(* Schneider Machine Expert - Basic project pick_place_SCADA, file version 2.7.0.0 *)
(* ProjectInformations: Name=New project *)

HARDWARE
  Cpu 0: TM221C16R
  EthernetConfiguration: NetworkName=M221, IpAllocationMode=FixedAddress, IpAddress=0.0.0.0, SubnetMask=0.0.0.0
  SerialLineConfiguration: Baud=Baud19200, Parity=ParityEven, DataBits=DataBits8, StopBits=StopBits1, PhysicalMedium=PhysicalMediumRs485, TransmissionMode=TransmissionModeModbusRtu, SlaveId=1, Addressing=SlaveAddressing
  MastTask: UsePeriodScanMode=false, PeriodScan=100
  FastTask: Period=255
  CpuBehavior: StartingMode=StartAsPreviousState, AutoSaveRamOnEeprom=true, WatchdogPeriod=250

SYMBOLS  (address, symbol, comment, settings)
  %M0       BOX_AT_PLACE
  %M1       PART_AT_PLACE
  %M2       DETECTED
  %M3       C_LIMIT
  %M4       START_
  %M5       RESET
  %M6       STOP
  %M7       EMERGENCY_STOP
  %M8       AUTO
  %M10      SENSOR_SALIDA
  %M20      BOX_CONVEYOR
  %M21      PART_CONVEYOR
  %M22      EXIT_CONVEYOR
  %M23      C_MAS
  %M24      GRAB
  %M25      EXIT_GREEN
  %M26      EXIT_YELLOW
  %M27      EXIT_RED
  %M28      START_LIGHT
  %M29      RESET_LIGHT
  %M30      STOP_LIGHT
  %M31      BOX_EMITTER
  %M32      PART_EMITTER
  %M33      FACTORY_RESET
  %M34      REMOVE
  %M50      GRAB_SCADA
  %M52      GIRO_ARDUINO
  %M54      STOP_ARDUINO
  %M56      RESET_ARDUINO
  %M60      E0
  %M61      E1
  %M62      E2
  %M63      E3
  %M64      E4
  %M65      E5
  %M66      E6
  %M67      E7
  %M68      E8
  %M69      E9
  %M70      E10
  %M71      E11
  %M72      E12
  %M77      E1_1
  %M80      E_MANUAL
  %M81      E3_1
  %M82      E7_1
  %M90      C1
  %M91      C2
  %MD0      X
  %MD2      Y
  %MD4      Z
  %MD10     SP_X
  %MD12     SP_Y
  %MD14     SP_Z
  %MD16     COUNTER
  %MD18     DISPLAY_PEDIDO
  %MD26     SP_X_ARDUINO
  %MD28     SP_Y_SCADA
  %MD30     SP_Z_SCADA
  %MD32     PEDIDO_ARDUINO
  %TM0      TON_1  [Preset=2, Base=OneSecond]
  %TM1      TON_2  [Preset=2, Base=OneSecond]
  %TM2      TON_3  [Preset=2, Base=OneSecond]
  %TM3        [Preset=1, Base=OneSecond]
  %TM4        [Preset=1, Base=OneSecond]
  %TM5        [Preset=3, Base=OneSecond]
  %TM6        [Preset=2, Base=OneSecond]
  %TM7        [Preset=2, Base=OneSecond]
  %TM8        [Preset=2, Base=OneSecond]

POU New POU
  (* SectionNumber=1 *)

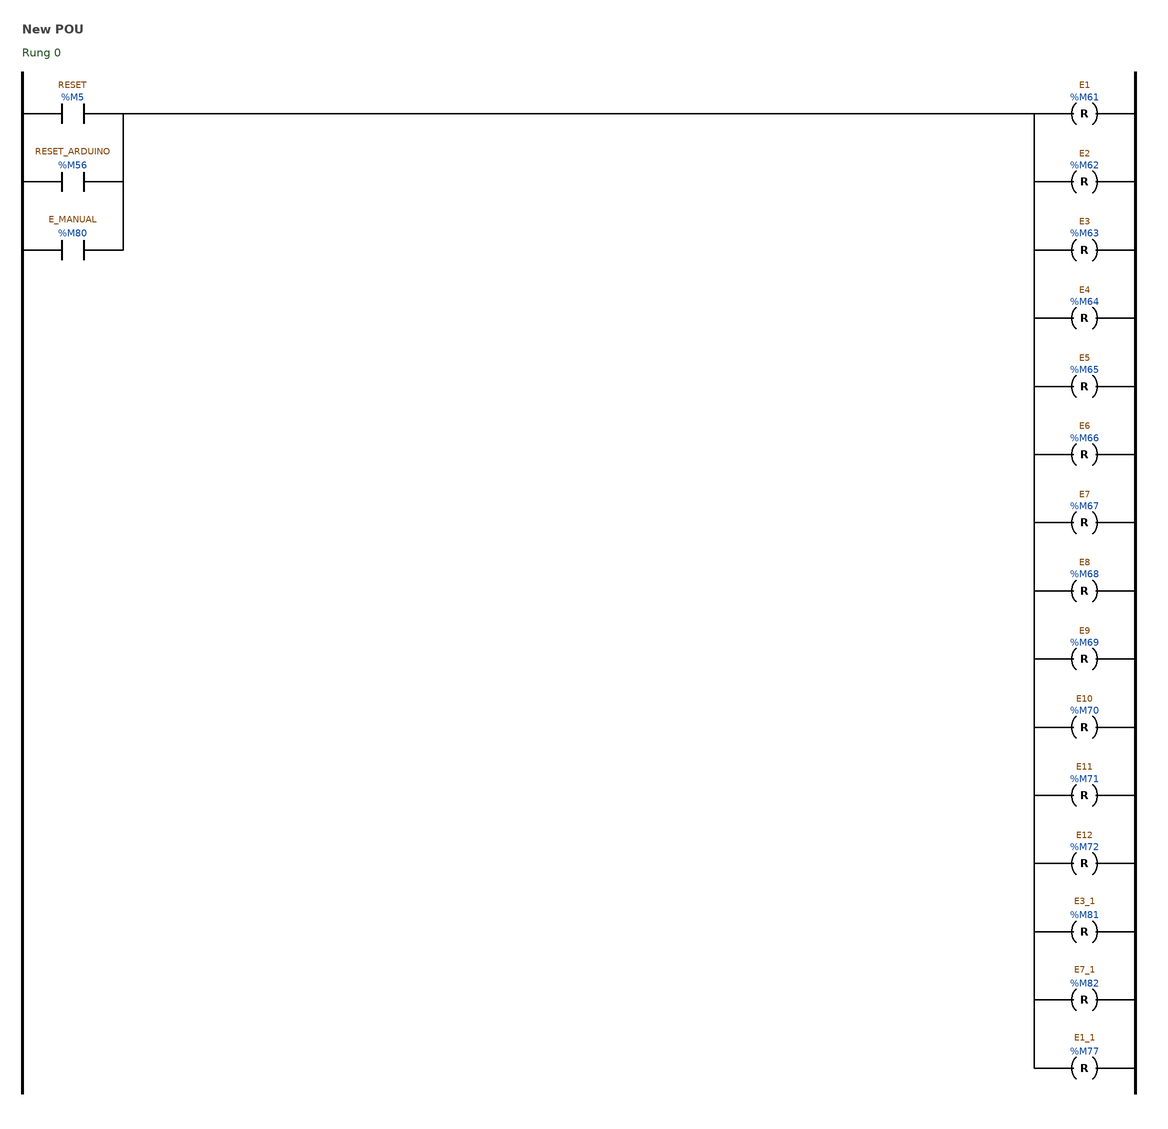

// Rung 0
  LD %M5                  (* RESET *)
  OR %M56                 (* RESET_ARDUINO *)
  OR %M80                 (* E_MANUAL *)
  R %M61                  (* E1 *)
  R %M62                  (* E2 *)
  R %M63                  (* E3 *)
  R %M64                  (* E4 *)
  R %M65                  (* E5 *)
  R %M66                  (* E6 *)
  R %M67                  (* E7 *)
  R %M68                  (* E8 *)
  R %M69                  (* E9 *)
  R %M70                  (* E10 *)
  R %M71                  (* E11 *)
  R %M72                  (* E12 *)
  R %M81                  (* E3_1 *)
  R %M82                  (* E7_1 *)
  R %M77                  (* E1_1 *)
  // as ST:
  //   IF RESET OR RESET_ARDUINO OR E_MANUAL THEN E1 := FALSE; END_IF;
  //   IF RESET OR RESET_ARDUINO OR E_MANUAL THEN E2 := FALSE; END_IF;
  //   IF RESET OR RESET_ARDUINO OR E_MANUAL THEN E3 := FALSE; END_IF;
  //   IF RESET OR RESET_ARDUINO OR E_MANUAL THEN E4 := FALSE; END_IF;
  //   IF RESET OR RESET_ARDUINO OR E_MANUAL THEN E5 := FALSE; END_IF;
  //   IF RESET OR RESET_ARDUINO OR E_MANUAL THEN E6 := FALSE; END_IF;
  //   IF RESET OR RESET_ARDUINO OR E_MANUAL THEN E7 := FALSE; END_IF;
  //   IF RESET OR RESET_ARDUINO OR E_MANUAL THEN E8 := FALSE; END_IF;
  //   IF RESET OR RESET_ARDUINO OR E_MANUAL THEN E9 := FALSE; END_IF;
  //   IF RESET OR RESET_ARDUINO OR E_MANUAL THEN E10 := FALSE; END_IF;
  //   IF RESET OR RESET_ARDUINO OR E_MANUAL THEN E11 := FALSE; END_IF;
  //   IF RESET OR RESET_ARDUINO OR E_MANUAL THEN E12 := FALSE; END_IF;
  //   IF RESET OR RESET_ARDUINO OR E_MANUAL THEN E3_1 := FALSE; END_IF;
  //   IF RESET OR RESET_ARDUINO OR E_MANUAL THEN E7_1 := FALSE; END_IF;
  //   IF RESET OR RESET_ARDUINO OR E_MANUAL THEN E1_1 := FALSE; END_IF;

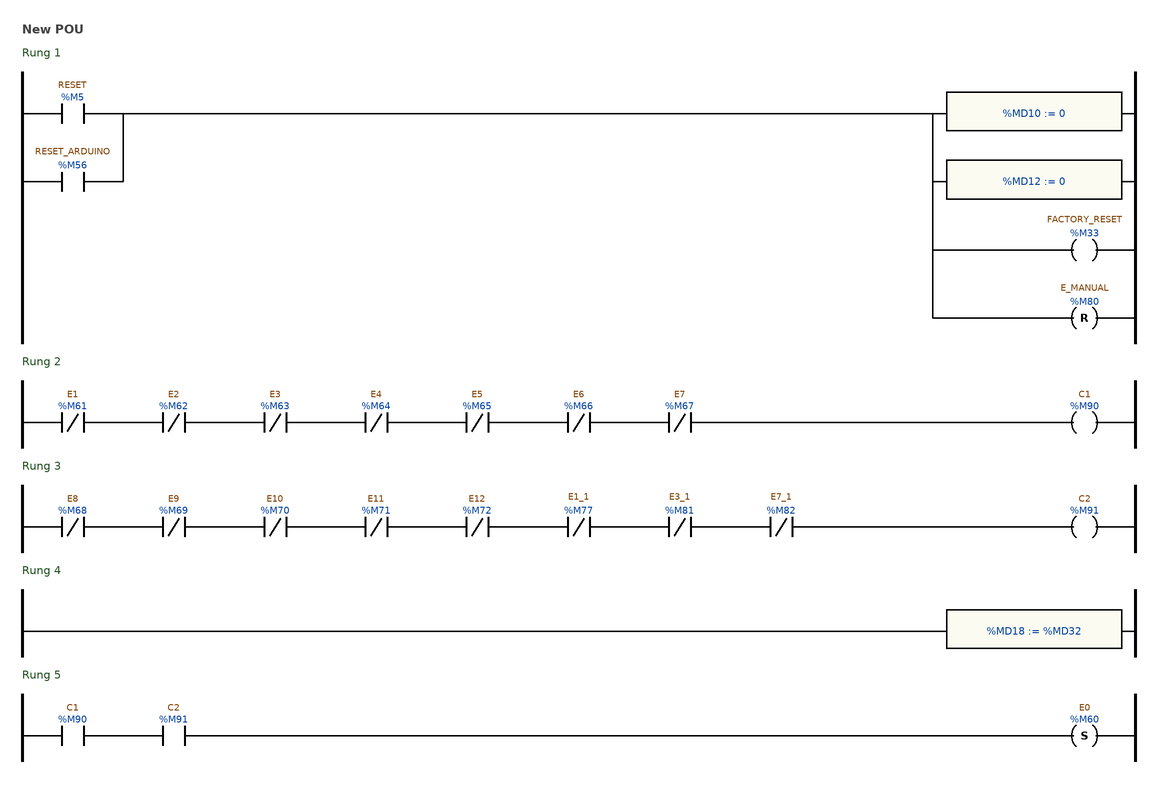

// Rung 1
  LD %M5                  (* RESET *)
  OR %M56                 (* RESET_ARDUINO *)
  [ %MD10 := 0 ]          (* SP_X *)
  [ %MD12 := 0 ]          (* SP_Y *)
  ST %M33                 (* FACTORY_RESET *)
  R %M80                  (* E_MANUAL *)
  // as ST:
  //   IF RESET OR RESET_ARDUINO THEN SP_X := 0; END_IF;
  //   IF RESET OR RESET_ARDUINO THEN SP_Y := 0; END_IF;
  //   FACTORY_RESET := RESET OR RESET_ARDUINO;
  //   IF RESET OR RESET_ARDUINO THEN E_MANUAL := FALSE; END_IF;

// Rung 2
  LDN %M61                (* E1 *)
  ANDN %M62               (* E2 *)
  ANDN %M63               (* E3 *)
  ANDN %M64               (* E4 *)
  ANDN %M65               (* E5 *)
  ANDN %M66               (* E6 *)
  ANDN %M67               (* E7 *)
  ST %M90                 (* C1 *)
  // as ST:
  //   C1 := NOT E1 AND NOT E2 AND NOT E3 AND NOT E4 AND NOT E5 AND NOT E6 AND NOT E7;

// Rung 3
  LDN %M68                (* E8 *)
  ANDN %M69               (* E9 *)
  ANDN %M70               (* E10 *)
  ANDN %M71               (* E11 *)
  ANDN %M72               (* E12 *)
  ANDN %M77               (* E1_1 *)
  ANDN %M81               (* E3_1 *)
  ANDN %M82               (* E7_1 *)
  ST %M91                 (* C2 *)
  // as ST:
  //   C2 := NOT E8 AND NOT E9 AND NOT E10 AND NOT E11 AND NOT E12 AND NOT E1_1 AND NOT E3_1 AND NOT E7_1;

// Rung 4
  LD 1
  [ %MD18 := %MD32 ]      (* DISPLAY_PEDIDO, PEDIDO_ARDUINO *)
  // as ST:
  //   DISPLAY_PEDIDO := PEDIDO_ARDUINO;

// Rung 5
  LD %M90                 (* C1 *)
  AND %M91                (* C2 *)
  S %M60                  (* E0 *)
  // as ST:
  //   IF C1 AND C2 THEN E0 := TRUE; END_IF;

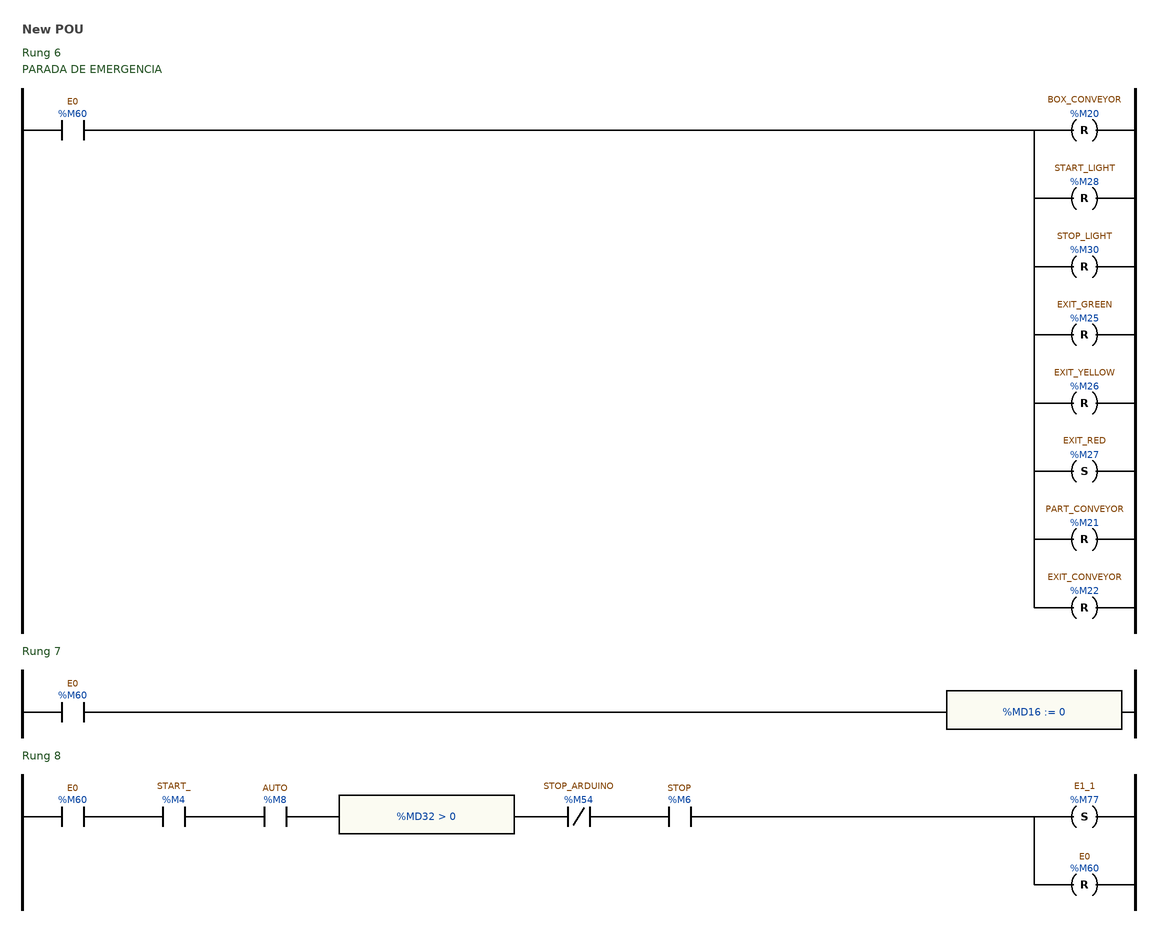

// Rung 6
// PARADA DE EMERGENCIA
  LD %M60                 (* E0 *)
  R %M20                  (* BOX_CONVEYOR *)
  R %M28                  (* START_LIGHT *)
  R %M30                  (* STOP_LIGHT *)
  R %M25                  (* EXIT_GREEN *)
  R %M26                  (* EXIT_YELLOW *)
  S %M27                  (* EXIT_RED *)
  R %M21                  (* PART_CONVEYOR *)
  R %M22                  (* EXIT_CONVEYOR *)
  // as ST:
  //   IF E0 THEN BOX_CONVEYOR := FALSE; END_IF;
  //   IF E0 THEN START_LIGHT := FALSE; END_IF;
  //   IF E0 THEN STOP_LIGHT := FALSE; END_IF;
  //   IF E0 THEN EXIT_GREEN := FALSE; END_IF;
  //   IF E0 THEN EXIT_YELLOW := FALSE; END_IF;
  //   IF E0 THEN EXIT_RED := TRUE; END_IF;
  //   IF E0 THEN PART_CONVEYOR := FALSE; END_IF;
  //   IF E0 THEN EXIT_CONVEYOR := FALSE; END_IF;

// Rung 7
  LD %M60                 (* E0 *)
  [ %MD16 := 0 ]          (* COUNTER *)
  // as ST:
  //   IF E0 THEN COUNTER := 0; END_IF;

// Rung 8
  LD %M60                 (* E0 *)
  AND %M4                 (* START_ *)
  AND %M8                 (* AUTO *)
  AND [ %MD32 > 0 ]       (* PEDIDO_ARDUINO *)
  ANDN %M54               (* STOP_ARDUINO *)
  AND %M6                 (* STOP *)
  S %M77                  (* E1_1 *)
  R %M60                  (* E0 *)
  // as ST:
  //   IF E0 AND START_ AND AUTO AND PEDIDO_ARDUINO > 0 AND NOT STOP_ARDUINO AND STOP THEN E1_1 := TRUE; END_IF;
  //   IF E0 AND START_ AND AUTO AND PEDIDO_ARDUINO > 0 AND NOT STOP_ARDUINO AND STOP THEN E0 := FALSE; END_IF;

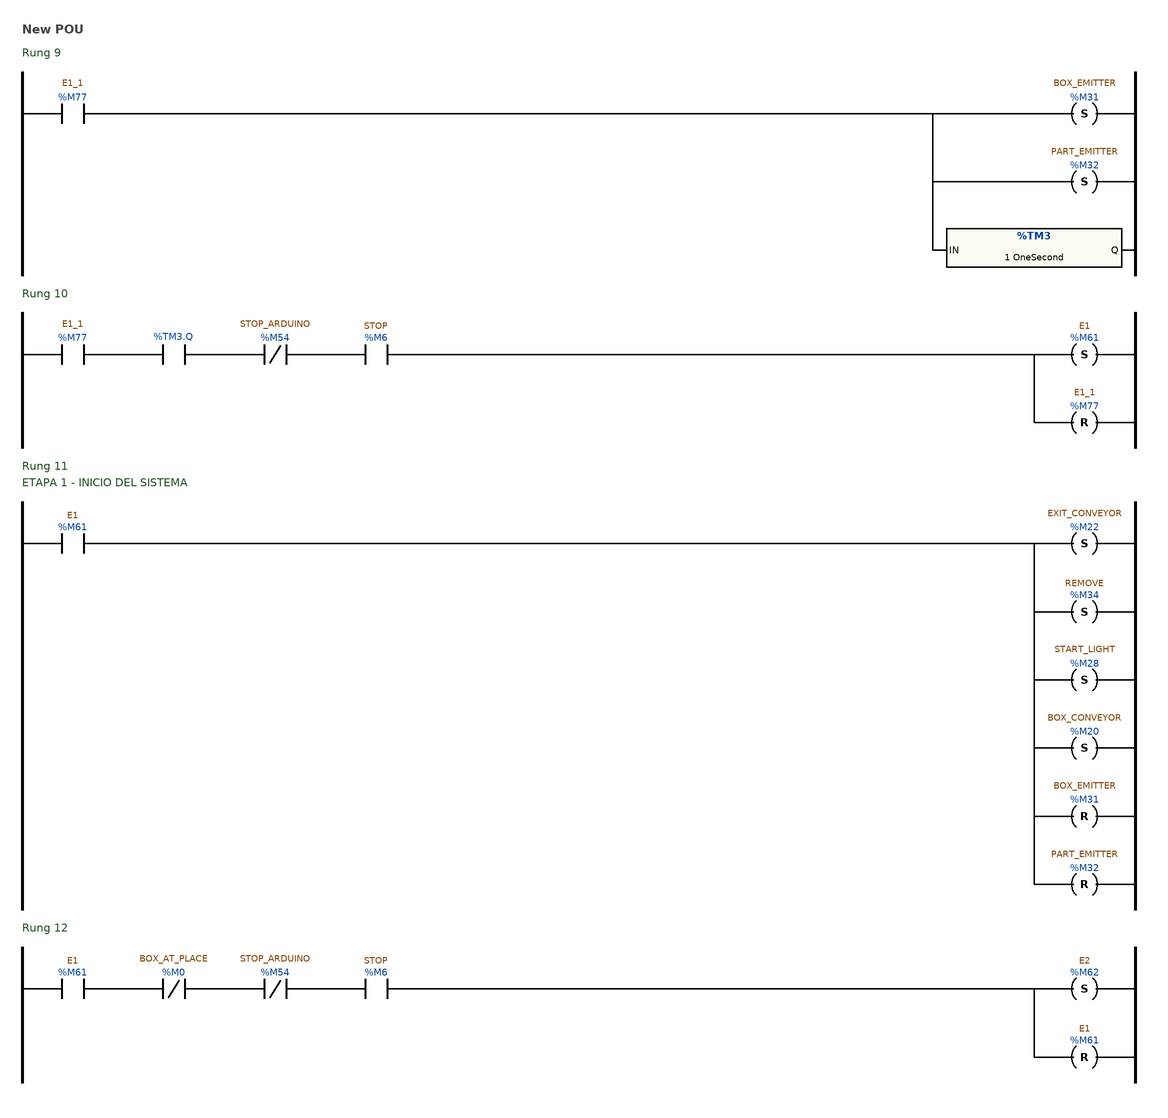

// Rung 9
  LD 1
  MULTIFB
  LD 1
  AND %M77                (* E1_1 *)
  ST %MW2009:X0
  LD %MW2009:X0
  S %M31                  (* BOX_EMITTER *)
  S %M32                  (* PART_EMITTER *)
  BLK %TM3
  LD %MW2009:X0
  IN
  END_BLK
  MULTIFB
  // as ST:
  //   IF E1_1 THEN BOX_EMITTER := TRUE; END_IF;
  //   IF E1_1 THEN PART_EMITTER := TRUE; END_IF;
  //   %TM3(IN := E1_1);

// Rung 10
  LD %M77                 (* E1_1 *)
  AND %TM3.Q
  ANDN %M54               (* STOP_ARDUINO *)
  AND %M6                 (* STOP *)
  S %M61                  (* E1 *)
  R %M77                  (* E1_1 *)
  // as ST:
  //   IF E1_1 AND %TM3.Q AND NOT STOP_ARDUINO AND STOP THEN E1 := TRUE; END_IF;
  //   IF E1_1 AND %TM3.Q AND NOT STOP_ARDUINO AND STOP THEN E1_1 := FALSE; END_IF;

// Rung 11
// ETAPA 1 - INICIO DEL SISTEMA
  LD %M61                 (* E1 *)
  S %M22                  (* EXIT_CONVEYOR *)
  S %M34                  (* REMOVE *)
  S %M28                  (* START_LIGHT *)
  S %M20                  (* BOX_CONVEYOR *)
  R %M31                  (* BOX_EMITTER *)
  R %M32                  (* PART_EMITTER *)
  // as ST:
  //   IF E1 THEN EXIT_CONVEYOR := TRUE; END_IF;
  //   IF E1 THEN REMOVE := TRUE; END_IF;
  //   IF E1 THEN START_LIGHT := TRUE; END_IF;
  //   IF E1 THEN BOX_CONVEYOR := TRUE; END_IF;
  //   IF E1 THEN BOX_EMITTER := FALSE; END_IF;
  //   IF E1 THEN PART_EMITTER := FALSE; END_IF;

// Rung 12
  LD %M61                 (* E1 *)
  ANDN %M0                (* BOX_AT_PLACE *)
  ANDN %M54               (* STOP_ARDUINO *)
  AND %M6                 (* STOP *)
  S %M62                  (* E2 *)
  R %M61                  (* E1 *)
  // as ST:
  //   IF E1 AND NOT BOX_AT_PLACE AND NOT STOP_ARDUINO AND STOP THEN E2 := TRUE; END_IF;
  //   IF E1 AND NOT BOX_AT_PLACE AND NOT STOP_ARDUINO AND STOP THEN E1 := FALSE; END_IF;

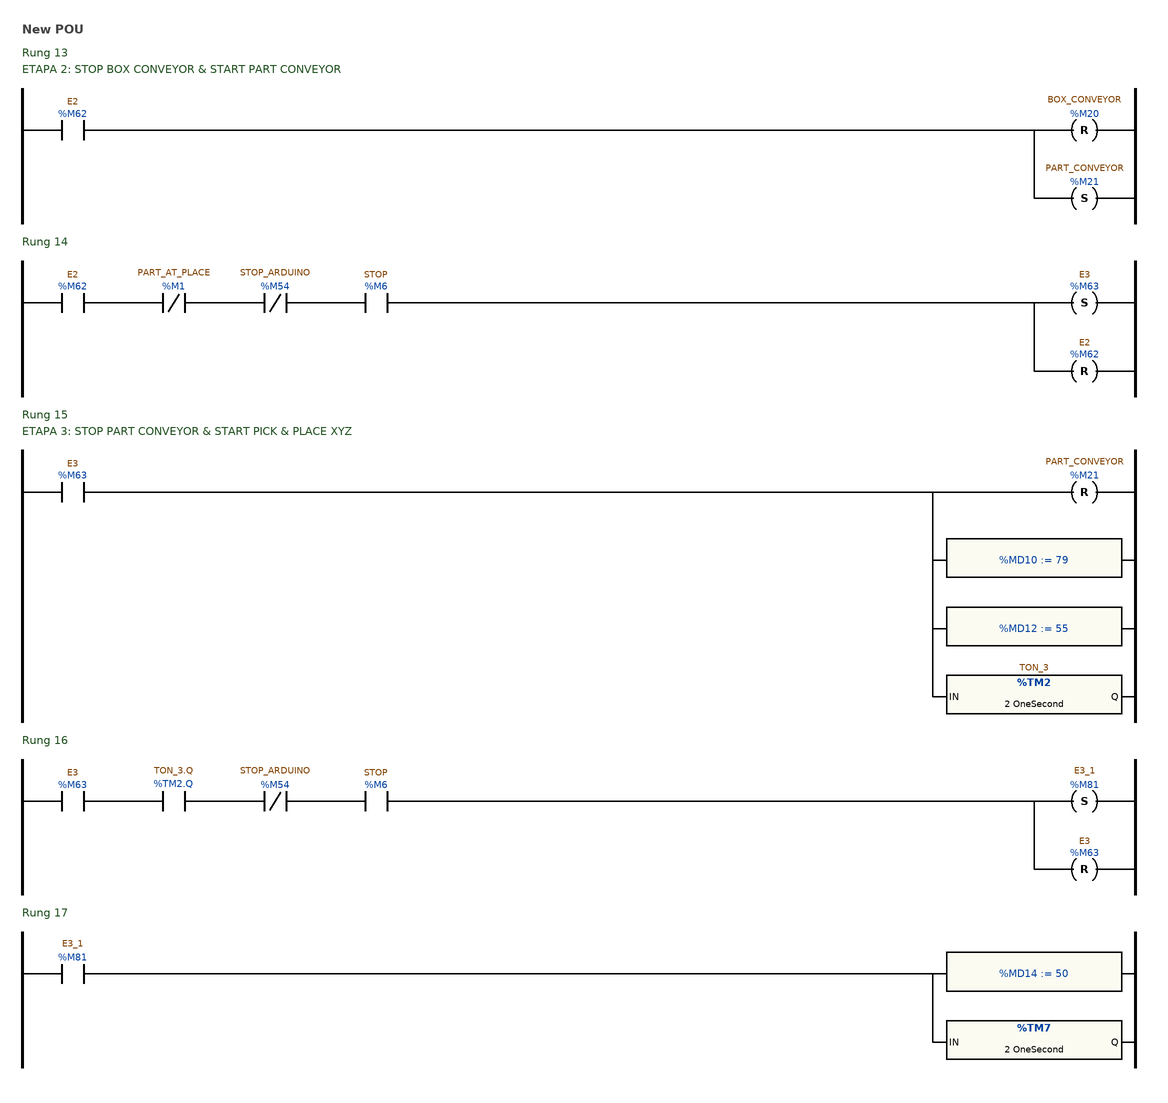

// Rung 13
// ETAPA 2: STOP BOX CONVEYOR & START PART CONVEYOR
  LD %M62                 (* E2 *)
  R %M20                  (* BOX_CONVEYOR *)
  S %M21                  (* PART_CONVEYOR *)
  // as ST:
  //   IF E2 THEN BOX_CONVEYOR := FALSE; END_IF;
  //   IF E2 THEN PART_CONVEYOR := TRUE; END_IF;

// Rung 14
  LD %M62                 (* E2 *)
  ANDN %M1                (* PART_AT_PLACE *)
  ANDN %M54               (* STOP_ARDUINO *)
  AND %M6                 (* STOP *)
  S %M63                  (* E3 *)
  R %M62                  (* E2 *)
  // as ST:
  //   IF E2 AND NOT PART_AT_PLACE AND NOT STOP_ARDUINO AND STOP THEN E3 := TRUE; END_IF;
  //   IF E2 AND NOT PART_AT_PLACE AND NOT STOP_ARDUINO AND STOP THEN E2 := FALSE; END_IF;

// Rung 15
// ETAPA 3: STOP PART CONVEYOR & START PICK & PLACE XYZ
  LD 1
  MULTIFB
  LD 1
  AND %M63                (* E3 *)
  ST %MW2009:X0
  LD %MW2009:X0
  R %M21                  (* PART_CONVEYOR *)
  [ %MD10 := 79 ]         (* SP_X *)
  [ %MD12 := 55 ]         (* SP_Y *)
  BLK %TM2                (* TON_3 *)
  LD %MW2009:X0
  IN
  END_BLK
  MULTIFB
  // as ST:
  //   IF E3 THEN PART_CONVEYOR := FALSE; END_IF;
  //   IF E3 THEN SP_X := 79; END_IF;
  //   IF E3 THEN SP_Y := 55; END_IF;
  //   TON_3(IN := E3);

// Rung 16
  LD %M63                 (* E3 *)
  AND %TM2.Q              (* TON_3 *)
  ANDN %M54               (* STOP_ARDUINO *)
  AND %M6                 (* STOP *)
  S %M81                  (* E3_1 *)
  R %M63                  (* E3 *)
  // as ST:
  //   IF E3 AND TON_3.Q AND NOT STOP_ARDUINO AND STOP THEN E3_1 := TRUE; END_IF;
  //   IF E3 AND TON_3.Q AND NOT STOP_ARDUINO AND STOP THEN E3 := FALSE; END_IF;

// Rung 17
  LD 1
  MULTIFB
  LD 1
  AND %M81                (* E3_1 *)
  ST %MW2009:X0
  LD %MW2009:X0
  [ %MD14 := 50 ]         (* SP_Z *)
  BLK %TM7
  LD %MW2009:X0
  IN
  END_BLK
  MULTIFB
  // as ST:
  //   IF E3_1 THEN SP_Z := 50; END_IF;
  //   %TM7(IN := E3_1);

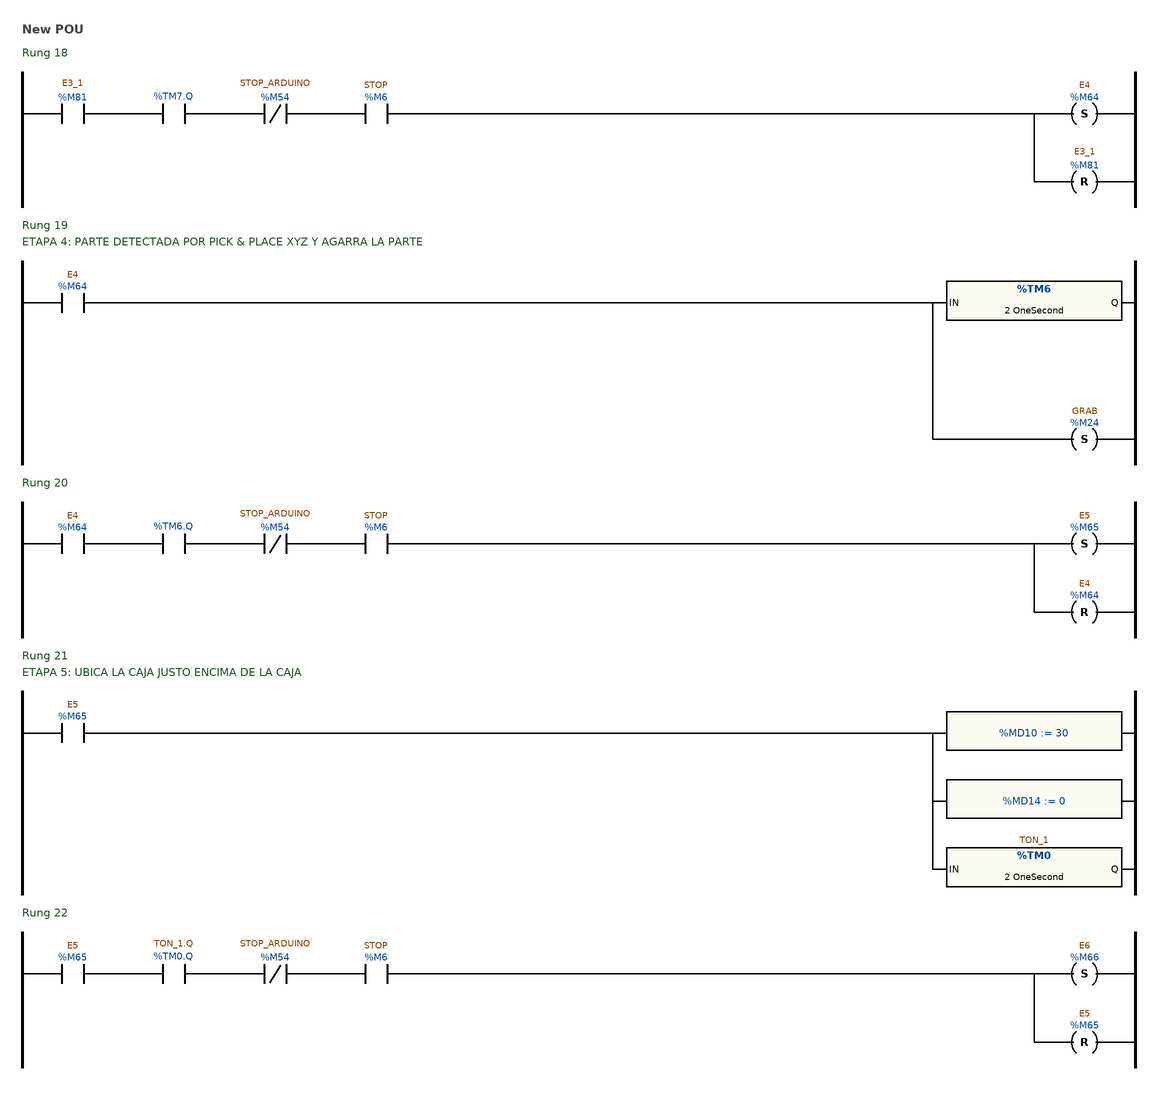

// Rung 18
  LD %M81                 (* E3_1 *)
  AND %TM7.Q
  ANDN %M54               (* STOP_ARDUINO *)
  AND %M6                 (* STOP *)
  S %M64                  (* E4 *)
  R %M81                  (* E3_1 *)
  // as ST:
  //   IF E3_1 AND %TM7.Q AND NOT STOP_ARDUINO AND STOP THEN E4 := TRUE; END_IF;
  //   IF E3_1 AND %TM7.Q AND NOT STOP_ARDUINO AND STOP THEN E3_1 := FALSE; END_IF;

// Rung 19
// ETAPA 4: PARTE DETECTADA POR PICK & PLACE XYZ Y AGARRA LA PARTE
  LD 1
  MULTIFB
  LD 1
  AND %M64                (* E4 *)
  ST %MW2009:X0
  BLK %TM6
  LD %MW2009:X0
  IN
  END_BLK
  LD %MW2009:X0
  S %M24                  (* GRAB *)
  MULTIFB
  // as ST:
  //   %TM6(IN := E4);
  //   IF E4 THEN GRAB := TRUE; END_IF;

// Rung 20
  LD %M64                 (* E4 *)
  AND %TM6.Q
  ANDN %M54               (* STOP_ARDUINO *)
  AND %M6                 (* STOP *)
  S %M65                  (* E5 *)
  R %M64                  (* E4 *)
  // as ST:
  //   IF E4 AND %TM6.Q AND NOT STOP_ARDUINO AND STOP THEN E5 := TRUE; END_IF;
  //   IF E4 AND %TM6.Q AND NOT STOP_ARDUINO AND STOP THEN E4 := FALSE; END_IF;

// Rung 21
// ETAPA 5: UBICA LA CAJA JUSTO ENCIMA DE LA CAJA
  LD 1
  MULTIFB
  LD 1
  AND %M65                (* E5 *)
  ST %MW2009:X0
  LD %MW2009:X0
  [ %MD10 := 30 ]         (* SP_X *)
  [ %MD14 := 0 ]          (* SP_Z *)
  BLK %TM0                (* TON_1 *)
  LD %MW2009:X0
  IN
  END_BLK
  MULTIFB
  // as ST:
  //   IF E5 THEN SP_X := 30; END_IF;
  //   IF E5 THEN SP_Z := 0; END_IF;
  //   TON_1(IN := E5);

// Rung 22
  LD %M65                 (* E5 *)
  AND %TM0.Q              (* TON_1 *)
  ANDN %M54               (* STOP_ARDUINO *)
  AND %M6                 (* STOP *)
  S %M66                  (* E6 *)
  R %M65                  (* E5 *)
  // as ST:
  //   IF E5 AND TON_1.Q AND NOT STOP_ARDUINO AND STOP THEN E6 := TRUE; END_IF;
  //   IF E5 AND TON_1.Q AND NOT STOP_ARDUINO AND STOP THEN E5 := FALSE; END_IF;

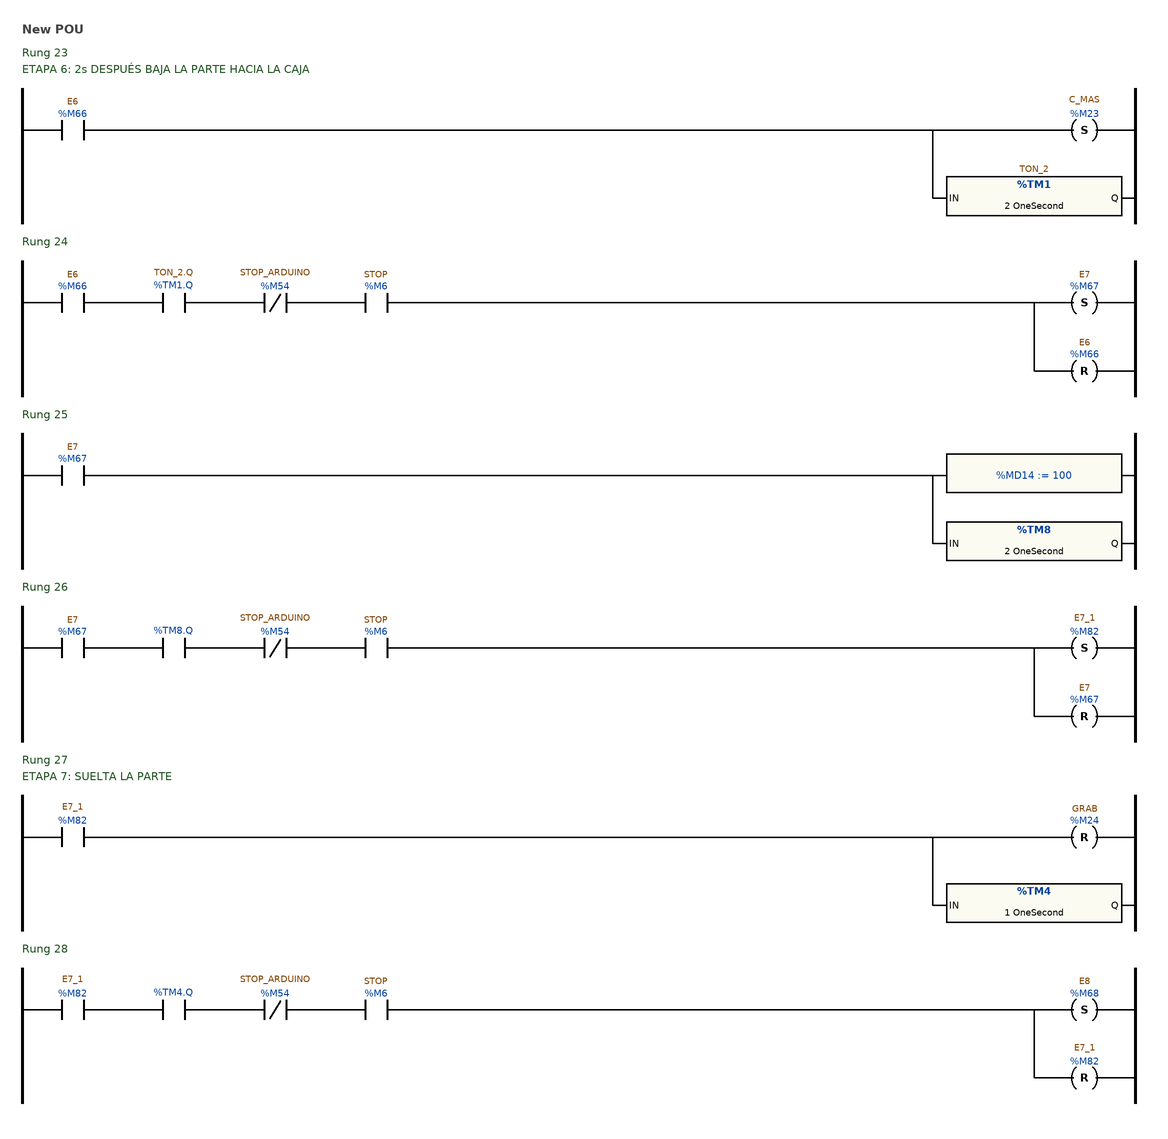

// Rung 23
// ETAPA 6: 2s DESPUÉS BAJA LA PARTE HACIA LA CAJA
  LD 1
  MULTIFB
  LD 1
  AND %M66                (* E6 *)
  ST %MW2009:X0
  LD %MW2009:X0
  S %M23                  (* C_MAS *)
  BLK %TM1                (* TON_2 *)
  LD %MW2009:X0
  IN
  END_BLK
  MULTIFB
  // as ST:
  //   IF E6 THEN C_MAS := TRUE; END_IF;
  //   TON_2(IN := E6);

// Rung 24
  LD %M66                 (* E6 *)
  AND %TM1.Q              (* TON_2 *)
  ANDN %M54               (* STOP_ARDUINO *)
  AND %M6                 (* STOP *)
  S %M67                  (* E7 *)
  R %M66                  (* E6 *)
  // as ST:
  //   IF E6 AND TON_2.Q AND NOT STOP_ARDUINO AND STOP THEN E7 := TRUE; END_IF;
  //   IF E6 AND TON_2.Q AND NOT STOP_ARDUINO AND STOP THEN E6 := FALSE; END_IF;

// Rung 25
  LD 1
  MULTIFB
  LD 1
  AND %M67                (* E7 *)
  ST %MW2009:X0
  LD %MW2009:X0
  [ %MD14 := 100 ]        (* SP_Z *)
  BLK %TM8
  LD %MW2009:X0
  IN
  END_BLK
  MULTIFB
  // as ST:
  //   IF E7 THEN SP_Z := 100; END_IF;
  //   %TM8(IN := E7);

// Rung 26
  LD %M67                 (* E7 *)
  AND %TM8.Q
  ANDN %M54               (* STOP_ARDUINO *)
  AND %M6                 (* STOP *)
  S %M82                  (* E7_1 *)
  R %M67                  (* E7 *)
  // as ST:
  //   IF E7 AND %TM8.Q AND NOT STOP_ARDUINO AND STOP THEN E7_1 := TRUE; END_IF;
  //   IF E7 AND %TM8.Q AND NOT STOP_ARDUINO AND STOP THEN E7 := FALSE; END_IF;

// Rung 27
// ETAPA 7: SUELTA LA PARTE
  LD 1
  MULTIFB
  LD 1
  AND %M82                (* E7_1 *)
  ST %MW2009:X0
  LD %MW2009:X0
  R %M24                  (* GRAB *)
  BLK %TM4
  LD %MW2009:X0
  IN
  END_BLK
  MULTIFB
  // as ST:
  //   IF E7_1 THEN GRAB := FALSE; END_IF;
  //   %TM4(IN := E7_1);

// Rung 28
  LD %M82                 (* E7_1 *)
  AND %TM4.Q
  ANDN %M54               (* STOP_ARDUINO *)
  AND %M6                 (* STOP *)
  S %M68                  (* E8 *)
  R %M82                  (* E7_1 *)
  // as ST:
  //   IF E7_1 AND %TM4.Q AND NOT STOP_ARDUINO AND STOP THEN E8 := TRUE; END_IF;
  //   IF E7_1 AND %TM4.Q AND NOT STOP_ARDUINO AND STOP THEN E7_1 := FALSE; END_IF;

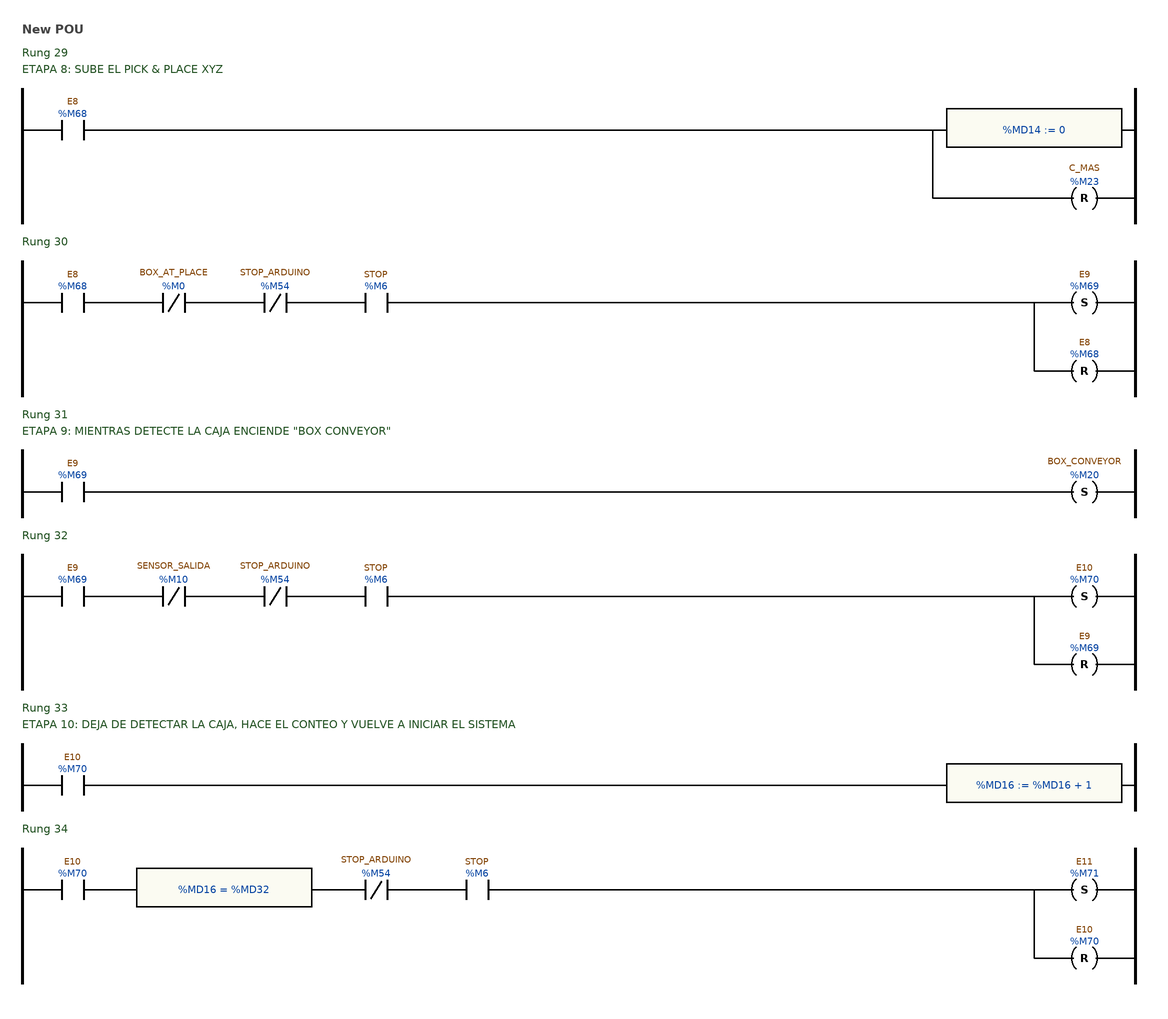

// Rung 29
// ETAPA 8: SUBE EL PICK & PLACE XYZ
  LD %M68                 (* E8 *)
  [ %MD14 := 0 ]          (* SP_Z *)
  R %M23                  (* C_MAS *)
  // as ST:
  //   IF E8 THEN SP_Z := 0; END_IF;
  //   IF E8 THEN C_MAS := FALSE; END_IF;

// Rung 30
  LD %M68                 (* E8 *)
  ANDN %M0                (* BOX_AT_PLACE *)
  ANDN %M54               (* STOP_ARDUINO *)
  AND %M6                 (* STOP *)
  S %M69                  (* E9 *)
  R %M68                  (* E8 *)
  // as ST:
  //   IF E8 AND NOT BOX_AT_PLACE AND NOT STOP_ARDUINO AND STOP THEN E9 := TRUE; END_IF;
  //   IF E8 AND NOT BOX_AT_PLACE AND NOT STOP_ARDUINO AND STOP THEN E8 := FALSE; END_IF;

// Rung 31
// ETAPA 9: MIENTRAS DETECTE LA CAJA ENCIENDE "BOX CONVEYOR"
  LD %M69                 (* E9 *)
  S %M20                  (* BOX_CONVEYOR *)
  // as ST:
  //   IF E9 THEN BOX_CONVEYOR := TRUE; END_IF;

// Rung 32
  LD %M69                 (* E9 *)
  ANDN %M10               (* SENSOR_SALIDA *)
  ANDN %M54               (* STOP_ARDUINO *)
  AND %M6                 (* STOP *)
  S %M70                  (* E10 *)
  R %M69                  (* E9 *)
  // as ST:
  //   IF E9 AND NOT SENSOR_SALIDA AND NOT STOP_ARDUINO AND STOP THEN E10 := TRUE; END_IF;
  //   IF E9 AND NOT SENSOR_SALIDA AND NOT STOP_ARDUINO AND STOP THEN E9 := FALSE; END_IF;

// Rung 33
// ETAPA 10: DEJA DE DETECTAR LA CAJA, HACE EL CONTEO Y VUELVE A INICIAR EL SISTEMA
  LD %M70                 (* E10 *)
  [ %MD16 := %MD16 + 1 ]  (* COUNTER, COUNTER *)
  // as ST:
  //   IF E10 THEN COUNTER := COUNTER + 1; END_IF;

// Rung 34
  LD %M70                 (* E10 *)
  AND [ %MD16 = %MD32 ]   (* COUNTER, PEDIDO_ARDUINO *)
  ANDN %M54               (* STOP_ARDUINO *)
  AND %M6                 (* STOP *)
  S %M71                  (* E11 *)
  R %M70                  (* E10 *)
  // as ST:
  //   IF E10 AND COUNTER = PEDIDO_ARDUINO AND NOT STOP_ARDUINO AND STOP THEN E11 := TRUE; END_IF;
  //   IF E10 AND COUNTER = PEDIDO_ARDUINO AND NOT STOP_ARDUINO AND STOP THEN E10 := FALSE; END_IF;

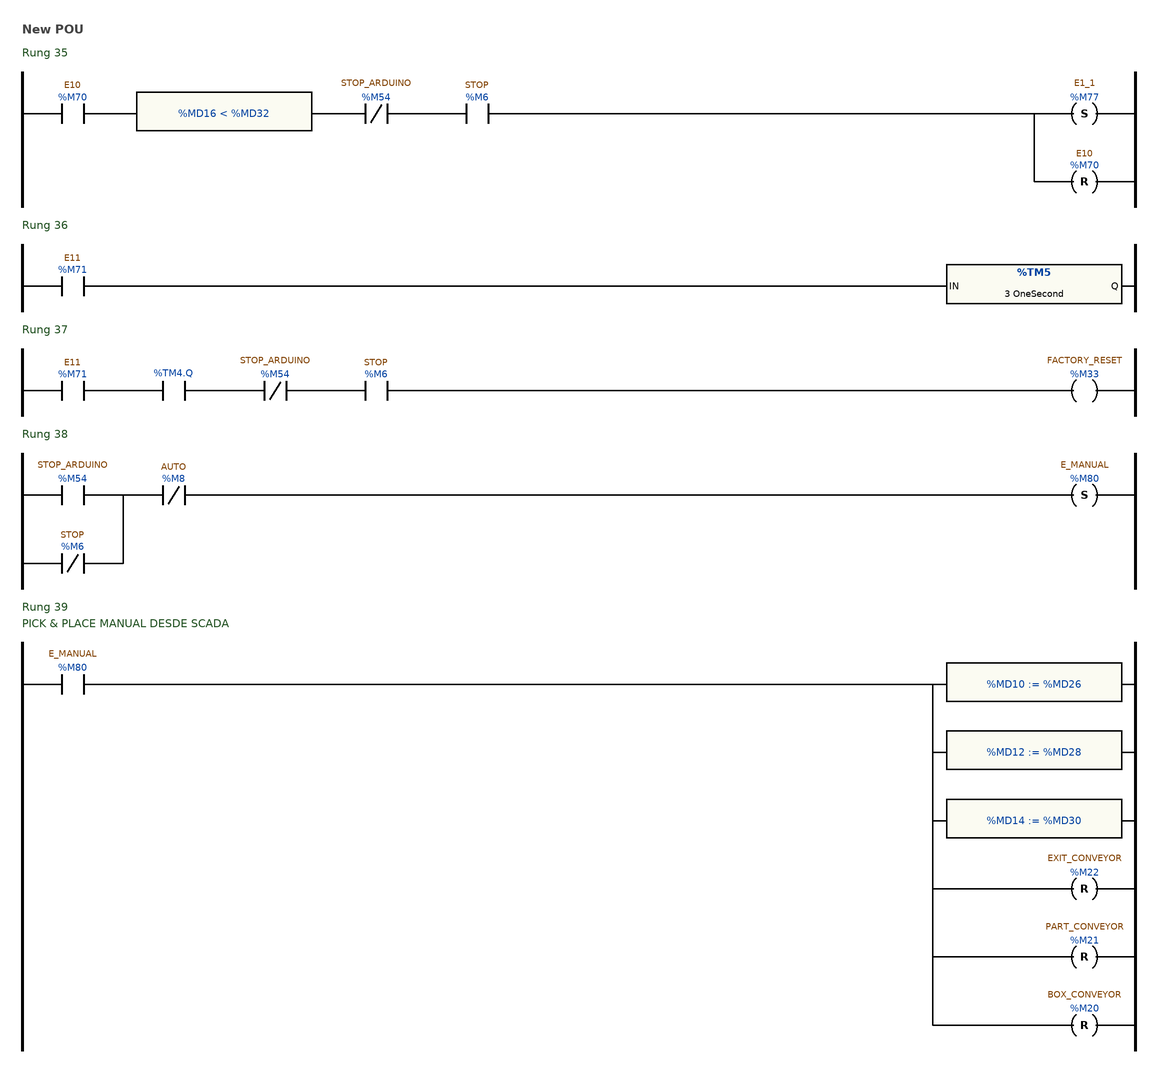

// Rung 35
  LD %M70                 (* E10 *)
  AND [ %MD16 < %MD32 ]   (* COUNTER, PEDIDO_ARDUINO *)
  ANDN %M54               (* STOP_ARDUINO *)
  AND %M6                 (* STOP *)
  S %M77                  (* E1_1 *)
  R %M70                  (* E10 *)
  // as ST:
  //   IF E10 AND COUNTER < PEDIDO_ARDUINO AND NOT STOP_ARDUINO AND STOP THEN E1_1 := TRUE; END_IF;
  //   IF E10 AND COUNTER < PEDIDO_ARDUINO AND NOT STOP_ARDUINO AND STOP THEN E10 := FALSE; END_IF;

// Rung 36
  BLK %TM5
  LD %M71                 (* E11 *)
  IN
  END_BLK
  // as ST:
  //   %TM5(IN := E11);

// Rung 37
  LD %M71                 (* E11 *)
  AND %TM4.Q
  ANDN %M54               (* STOP_ARDUINO *)
  AND %M6                 (* STOP *)
  ST %M33                 (* FACTORY_RESET *)
  // as ST:
  //   FACTORY_RESET := E11 AND %TM4.Q AND NOT STOP_ARDUINO AND STOP;

// Rung 38
  LD %M54                 (* STOP_ARDUINO *)
  ORN %M6                 (* STOP *)
  ANDN %M8                (* AUTO *)
  S %M80                  (* E_MANUAL *)
  // as ST:
  //   IF (STOP_ARDUINO OR NOT STOP) AND NOT AUTO THEN E_MANUAL := TRUE; END_IF;

// Rung 39
// PICK & PLACE MANUAL DESDE SCADA
  LD %M80                 (* E_MANUAL *)
  [ %MD10 := %MD26 ]      (* SP_X, SP_X_ARDUINO *)
  [ %MD12 := %MD28 ]      (* SP_Y, SP_Y_SCADA *)
  [ %MD14 := %MD30 ]      (* SP_Z, SP_Z_SCADA *)
  R %M22                  (* EXIT_CONVEYOR *)
  R %M21                  (* PART_CONVEYOR *)
  R %M20                  (* BOX_CONVEYOR *)
  // as ST:
  //   IF E_MANUAL THEN SP_X := SP_X_ARDUINO; END_IF;
  //   IF E_MANUAL THEN SP_Y := SP_Y_SCADA; END_IF;
  //   IF E_MANUAL THEN SP_Z := SP_Z_SCADA; END_IF;
  //   IF E_MANUAL THEN EXIT_CONVEYOR := FALSE; END_IF;
  //   IF E_MANUAL THEN PART_CONVEYOR := FALSE; END_IF;
  //   IF E_MANUAL THEN BOX_CONVEYOR := FALSE; END_IF;

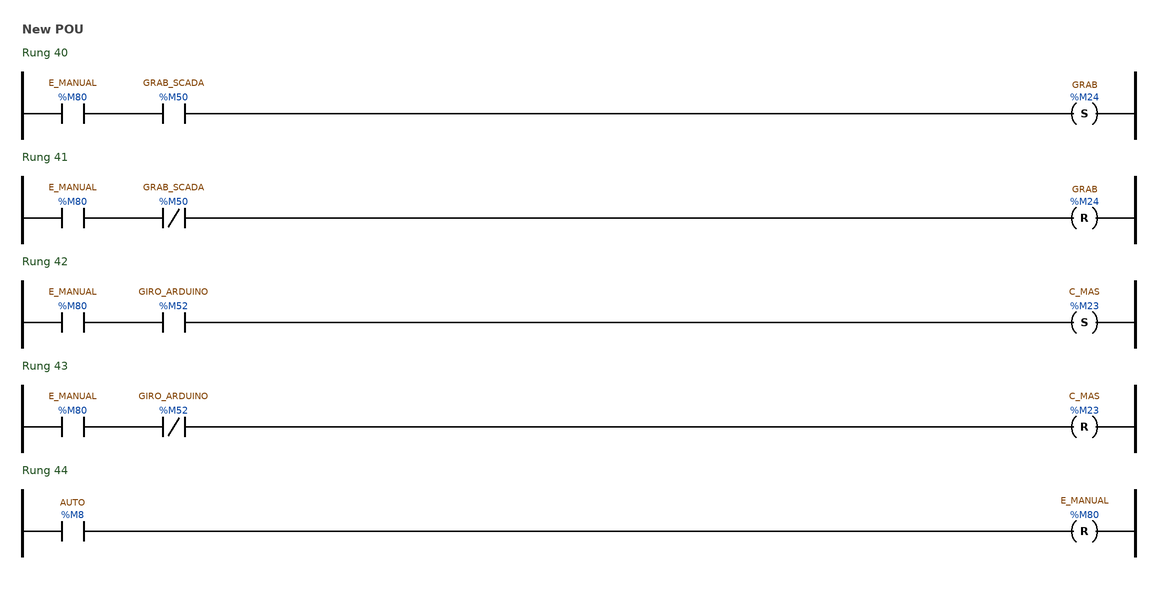

// Rung 40
  LD %M80                 (* E_MANUAL *)
  AND %M50                (* GRAB_SCADA *)
  S %M24                  (* GRAB *)
  // as ST:
  //   IF E_MANUAL AND GRAB_SCADA THEN GRAB := TRUE; END_IF;

// Rung 41
  LD %M80                 (* E_MANUAL *)
  ANDN %M50               (* GRAB_SCADA *)
  R %M24                  (* GRAB *)
  // as ST:
  //   IF E_MANUAL AND NOT GRAB_SCADA THEN GRAB := FALSE; END_IF;

// Rung 42
  LD %M80                 (* E_MANUAL *)
  AND %M52                (* GIRO_ARDUINO *)
  S %M23                  (* C_MAS *)
  // as ST:
  //   IF E_MANUAL AND GIRO_ARDUINO THEN C_MAS := TRUE; END_IF;

// Rung 43
  LD %M80                 (* E_MANUAL *)
  ANDN %M52               (* GIRO_ARDUINO *)
  R %M23                  (* C_MAS *)
  // as ST:
  //   IF E_MANUAL AND NOT GIRO_ARDUINO THEN C_MAS := FALSE; END_IF;

// Rung 44
  LD %M8                  (* AUTO *)
  R %M80                  (* E_MANUAL *)
  // as ST:
  //   IF AUTO THEN E_MANUAL := FALSE; END_IF;
